{attribute 'GeneratedUsingTerminal: EK1960-0000-0021'}
{attribute addProperty BoxType "EK1960-0000-0021"}
{attribute addProperty Id "OutputsOutputs_D994E0F924"}
{attribute addProperty CRC "2340071586"}
{attribute addProperty Size "24"}
TYPE Module_2_FSOUT_8B7AA8A2 :
STRUCT
	{attribute addProperty Name "Outputs"}
	Outputs  : Outputs_D994E0F9;
END_STRUCT
END_TYPE

(* stored: Version 1.2.0.0, ProductVersion 3.1.4024.9
   DUT Module_2_FSOUT_8B7AA8A2: Id {ac551d56-bd3e-4512-9efd-391b70c628f4} *)
